FUNCTION_BLOCK StartProgramTask EXTENDS TcoMitsubishiRoboticsTask
VAR

	_stopType: TcoAbstractions.eTcoRoboticsStopType;
END_VAR



IF Execute() THEN
	_blink(inOnTime:=T#500MS,inOffTime:=T#500MS);

	IF _progress = 0 THEN
		IF NOT __ISVALIDREF(inoControl) THEN
			_varInfo :=__VARINFO(inoControl);
			Messenger.Programming(_sb.Clear().Append('<#Invalid reference: #>').Append(_varInfo.Symbol).ToString()).Pin();
		ELSIF NOT __ISVALIDREF(inoConfig) THEN                                                  
			_varInfo :=__VARINFO(inoConfig);                                                    
			Messenger.Programming(_sb.Clear().Append('<#Invalid reference: #>').Append(_varInfo.Symbol).ToString()).Pin();
		ELSIF NOT __ISVALIDREF(inoStatus) THEN                                                  
			_varInfo :=__VARINFO(inoStatus);                                                    
			Messenger.Programming(_sb.Clear().Append('<#Invalid reference: #>').Append(_varInfo.Symbol).ToString()).Pin();
			ELSE
			_progress := _progress + 1;
		END_IF

	END_IF
	IF _progress = 1 THEN
		inoControl.OpoerationEnable:=TRUE;
		_varInfo :=__VARINFO( inoStatus.State.OperationEnable);                                                
		THIS^.Messenger.OnCondition(_infoTimer.Q AND NOT inoStatus.State.OperationEnable).Warning(_sb.Clear().Append('<#Waiting for Operation enable signal! #>').Append(_varInfo.Symbol).ToString());
		IF  inoStatus.State.OperationEnable THEN
			_progress := _progress + 1;
		END_IF;
	END_IF;
	
	IF _progress = 2 THEN
	
		inoControl.AutoEnable:=TRUE;
		_varInfo :=__VARINFO( inoStatus.State.AutoEnable);                                                
		THIS^.Messenger.OnCondition(_infoTimer.Q AND NOT inoStatus.State.AutoEnable).Warning(_sb.Clear().Append('<#Waiting for Auto signal! #>').Append(_varInfo.Symbol).ToString());
		IF  inoStatus.State.AutoEnable THEN
			_progress := _progress + 1;
		END_IF;
	END_IF;
	
	
	IF _progress =3 THEN	
		Messenger.Debug('<#Robot Error Reset#>');
		inoControl.ErrorReset := inoStatus.State.ErrorReset AND _blink.outQ;
		IF NOT inoStatus.State.ErrorReset THEN
			inoControl.ErrorReset:=FALSE;
			_progress := _progress + 1;
		END_IF
	END_IF;
	
	IF _progress = 4 THEN
		IF inoStatus.State.HighLevelError OR inoStatus.State.LowLevelError OR inoStatus.State.CautionLevelError OR  inoStatus.State.EmergencyError THEN 
			_progress := 1;
		END_IF
		inoControl.Start:=_blink.outQ;
		_varInfo :=__VARINFO( inoStatus.State.Start);                                                
		THIS^.Messenger.OnCondition(_infoTimer.Q AND NOT inoStatus.State.Start).Warning(_sb.Clear().Append('<#Waiting for program running signal! #>').Append(_varInfo.Symbol).ToString());
		
				
		IF  inoStatus.State.Start AND NOT inoStatus.State.ErrorReset THEN
				inoControl.Start:=FALSE;
		END_IF
	END_IF;		
	
	

    DoneWhen(inoStatus.State.Start AND NOT inoStatus.State.ErrorReset );
    CallTimers(TRUE);
	
	THIS^.ThrowWhen(_errorTimer.Q OR inoStatus.State.ErrorReset);
END_IF

IF  THIS^.Error AND NOT _errorMessage.Pinned THEN
	THIS^.Restore();
END_IF

METHOD PUBLIC FB_init : BOOL
VAR_INPUT
    bInitRetains : BOOL; // if TRUE, the retain variables are initialized (warm start / cold start)
    bInCopyCode : BOOL; // if TRUE, the instance afterwards gets moved into the copy code (online change)
  	ParentObject : ITcoObject;	
END_VAR
END_METHOD

METHOD INTERNAL InvokeWithParams : ITcoTaskStatus
VAR_INPUT
	inStopType : eTcoRoboticsStopType;
END_VAR
_stopType := inStopType;
InvokeWithParams := THIS^.Invoke();
END_METHOD

(*~
	<docu>
		<summary>
			Executes when task is aborted.
		</summary>			
	</docu>	
~*)
METHOD PROTECTED OnAbort
IF  __ISVALIDREF(inoStatus) THEN   THIS^.inoStatus.ActionDescription := '<#Stop program was aborted, while not yet completed!#>';END_IF;
END_METHOD

(*~
	<docu>
		<summary>
			Executes when task reaches the ```Done``` state .
		</summary>			
	</docu>	
~*)
METHOD PROTECTED OnDone
IF  __ISVALIDREF(inoStatus) THEN  THIS^.inoStatus.ActionDescription := '<#Stop program was completed successfully.#>';END_IF; 
_progress:=0;
END_METHOD

(*~
	<docu>
		<summary>
			Executes when task reaches the ```Error``` state.
				</summary>			
	</docu>	
~*)
METHOD PROTECTED OnError
VAR
	description: STRING;
END_VAR
THIS^.inoStatus.ActionDescription := '<#Stopping program with error.#>'; 
IF  __ISVALIDREF(inoStatus) THEN   THIS^.inoStatus.ActionDescription := description; END_IF;
THIS^._errorMessage.Error(_sb.Clear().Append(description).Append(' To restore acknowledge this alarm.').ToString()).Pin();
END_METHOD

METHOD PROTECTED OnStart
IF  __ISVALIDREF(inoStatus) THEN  THIS^.inoStatus.ActionDescription := '<#Stopping program started.#>'; END_IF; 
CallTimers(FALSE);
END_METHOD

(*~
	<docu>
		<summary>
			Restores this instance to the Ready state. Can be called explicitly or from within one of the restore mechanisms.
			<para>
				See also <see cref="PlcDocu.TcoCore.TcoTask.AutoRestorable()"/>
			</para>
		</summary>			
	</docu>	
~*)
METHOD Restore : ITcoRestorable
SUPER^.Restore();
END_METHOD

END_FUNCTION_BLOCK

(* stored: Version 1.1.0.1, ProductVersion 3.1.4024.12
   POU StartProgramTask: Id {7004f61d-cd33-02af-01b2-f630f74c88c6}, SpecialFunc None
   Method FB_init: Id {3251f34a-c5b5-0759-2786-4c5a4d33307a}
   Method InvokeWithParams: Id {c86c3fbb-f2f9-0b22-2eca-016e48529d36}
   Method OnAbort: Id {6fc5c01a-0e54-0761-1e35-310f3ecf8d57}
   Method OnDone: Id {d0836687-8734-03e6-2b24-e436e5af2908}
   Method OnError: Id {2144eadb-3cca-0716-3852-9cc611e2f12e}
   Method OnStart: Id {f73e3142-106e-0c6b-028d-d730ee2ea835}
   Method Restore: Id {88c8f898-59d3-0ecb-043e-38a3460f1709} *)
